{attribute 'linkalways'} 
{attribute 'no_explicit_call' := 'This FB is a CLASS and must be accessed using methods or properties'}
{attribute 'enable_dynamic_creation'}
FUNCTION_BLOCK LinkedListForwardEnumerator EXTENDS Disposable IMPLEMENTS I_ForwardEnumerator, I_EventHandler
VAR
	parent : I_LinkedList;
	currentNode : I_LinkedListNode;
	moveNextCalled : BOOL := FALSE;
	invalid : BOOL := FALSE; 
END_VAR

METHOD FB_init : BOOL
VAR_INPUT
	bInitRetains : BOOL; // if TRUE, the retain variables are initialized (warm start / cold start)
	bInCopyCode : BOOL;  // if TRUE, the instance afterwards gets moved into the copy code (online change)
	Parent : I_LinkedList;
END_VAR
Parent.OnEvent('OnLinkListChanged',THIS^);
this^.parent := Parent;
END_METHOD

METHOD PUBLIC Get : BOOL;
VAR_INPUT
	Destination : ANY;
END_VAR
IF currentNode <> 0 THEN
	Get := currentNode.Get(Destination);
END_IF
END_METHOD

METHOD PUBLIC GetTo : BOOL;
VAR_INPUT
	Destination : PVOID;
	DestinationSize : UDINT;
END_VAR
IF currentNode <> 0 THEN
	GetTo := currentNode.GetTo(Destination,DestinationSize);
END_IF
END_METHOD

METHOD PUBLIC HandleEvent
VAR_INPUT
	Event : I_Event;
END_VAR
VAR
	linkedListChangedEvent : I_LinkedListChangedEvent;
END_VAR
IF __QUERYINTERFACE(Event, linkedListChangedEvent) THEN
	invalid := TRUE;
	currentNode := 0;
END_IF
END_METHOD

PROPERTY PUBLIC IsValid : BOOL
GET
IsValid := not invalid;
END_GET
END_PROPERTY

METHOD PUBLIC MoveNext : BOOL
VAR_INPUT
END_VAR
IF invalid THEN
	RETURN;
END_IF

IF NOT moveNextCalled THEN
	moveNextCalled := TRUE;
	MoveNext := TRUE;	
	currentNode := parent.First;
	RETURN;
END_IF

IF currentNode = 0 THEN
	RETURN;
END_IF

if currentNode.Next <> 0 then
	currentNode := currentNode.Next;
	MoveNext := TRUE;	
	RETURN;
END_IF
END_METHOD

METHOD PROTECTED OnDispose : BOOL
VAR_INPUT
	CalledExplicitly : BOOL;
END_VAR
parent.OffEvent('OnLinkListChanged',this^);
END_METHOD

METHOD PUBLIC Reset
VAR_INPUT
END_VAR
currentNode := 0;
moveNextCalled := FALSE;
invalid := FALSE;
END_METHOD

END_FUNCTION_BLOCK

(* stored: Version 1.1.0.1, ProductVersion 3.1.4024.12
   POU LinkedListForwardEnumerator: Id {b1356522-2356-47f0-8fc3-88d40e839155}, SpecialFunc None
   Folder Constructor: Id {ba00adcc-08d5-4221-8a6d-f1cc9ae85243}
   Folder Protected: Id {d11b83b0-e836-463b-a509-88d4395e1f4f}
   Method FB_init: Id {9785a5f6-7e4a-4ea0-9517-538d8da73e6a}
   Method Get: Id {00128fb3-0888-4680-baae-fe94bc38c29b}
   Method GetTo: Id {1412ae45-9668-4dda-b44d-6048d41a0a8b}
   Method HandleEvent: Id {9b82c3a0-a8d9-4f44-aa61-0031448f4819}
   Property IsValid: Id {aff8eea1-92fe-4c1a-ab72-6d68ef134bd6}
   Get Get: Id {d7fac01e-4fea-4838-8ffe-61ec719ff66c}
   Method MoveNext: Id {6be4d0d4-bc06-473d-8ec1-a047989792d6}
   Method OnDispose: Id {57098a64-7040-4a4c-ad76-d4e0094e1750}
   Method Reset: Id {2017d8bc-6ce2-45f9-b0d2-516b5a2f274c} *)
